// SIMATIC STEP 7 (V5.x) project BOTTLING_PLANT
// station: Hardware
// station: SIMATIC 300(1)
// station: P_ADR_BUS

SYMBOL_TABLE
"BOTTELING PLANT"	FB 1	FB 1
"BOTTLE_MOVE"	FC 1	FC 1
"BOTTLE_FILL_MOVE"	FC 2	FC 2
"Tank_Filling"	FC 3	FC 3
"START"	I 0.0	BOOL
"LEVEL_HIGH"	I 0.1	BOOL
"LEVEL_LOW"	I 0.2	BOOL
"BOTTEL_PRESENT"	I 0.3	BOOL
"BOTTLE_FILLED"	I 0.4	BOOL
"I0.5"	I 0.5	BOOL
"MOTOR_SET_M"	M 0.2	BOOL
"BOTTEL_FILL_SNSED"	M 0.3	BOOL
"MOTOR_RESET_M"	M 0.4	BOOL
"LOW_LEVEL"	M 0.6	BOOL
"STOP"	M 1.3	BOOL
"TF_LL_CNT_BIT"	M 2.1	BOOL
"M_BOTTLE_PRE"	M 2.3	BOOL
"TF_SR_BIT"	M 4.5	BOOL
"EMG"	M 5.1	BOOL
"M"	MW 100	WORD
"V1"	Q 0.0	BOOL
"V2"	Q 0.1	BOOL
"MOTOR"	Q 0.2	BOOL
END_SYMBOL_TABLE
